// TIA Portal V20 export
TYPE "typeCmControlNodeInterlock"
// stored: Namespace Unit1.Em8
   STRUCT
      thicknessAxisZ : "LER_typeAxisInterlock";
      hipotThicknessServoPress : "LER_typeServoPressInterlock";
      hipotThicknessStageLiftFront : "LER_typeTwoWayActuatorInterlock";
      hipotThicknessStageLiftRear : "LER_typeTwoWayActuatorInterlock";
      hipotTabContactor : "LER_typeTwoWayActuatorInterlock";
      hipotTabContactorLeft : "LER_typeTwoWayActuatorInterlock";
      hipotTabContactorRight : "LER_typeTwoWayActuatorInterlock";
      hipotThicknessStageLiftAll : "LER_typeTwoWayActuatorInterlock";
   END_STRUCT;
END_TYPE
